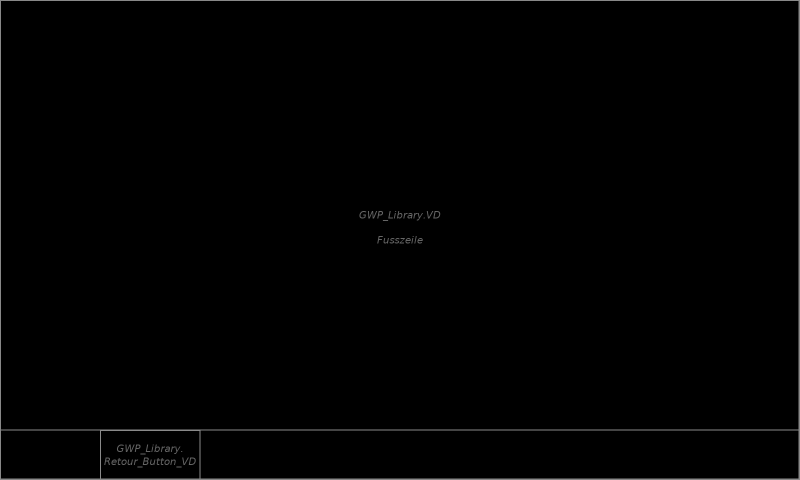
VISUALIZATION VD  // 800x480
    Frame (0,0 800x480)
        shows Fusszeile()
    Frame (100,430 100x50)
        shows GWP_Library.Retour_Button_VD()
    Frame (0,0 800x430)
        shows GWP_Library.VD(FB_VD := MAIN.VD_0)
END_VISUALIZATION

(* stored: Version 1.1.0.1, ProductVersion 3.1.4022.6
   Visu VD: Id {b1f8c38e-c24b-4e18-aa91-d5469a42ce00} *)
